// TIA Portal V17 export
// export: Created 2022-07-20T07:02:32.1719581Z, ExportSetting WithDefaults, DisplayName Totally Integrated Automation Portal, DisplayVersion V17, DisplayName TIA Portal Openness, DisplayVersion V17, DisplayName TIA Portal Version Control Interface, DisplayVersion V17, DisplayName SINAMICS Startdrive Advanced, DisplayVersion V17, DisplayName SINAMICS Startdrive G130, G150, S120, S150, SINAMICS MV, S210, DisplayVersion V17, DisplayName SINAMICS Startdrive G110M, G120, G120C, G120D, G120P, G115D, DisplayVersion V17, DisplayName STEP 7 Professional, DisplayVersion V17, DisplayName STEP 7 Safety, DisplayVersion V17, DisplayName WinCC Advanced, DisplayVersion V17
FUNCTION_BLOCK "FB11008_CamTrack"   // FB11008, LAD
{ S7_Optimized_Access := 'TRUE' }
VERSION : 0.1
// stored: AutoNumber false, IsIECCheckEnabled false, IsRetainMemResEnabled false, MemoryReserve 100, SetENOAutomatically false, UDAEnableTagReadback false
   VAR_INPUT
      Enable { ExternalAccessible := 'False'; ExternalVisible := 'False'; ExternalWritable := 'False'} : Bool;
      Cam { ExternalAccessible := 'False'; ExternalVisible := 'False'; ExternalWritable := 'False'} : Array[1..32] of TO_CamTrack_Struct_CamData;
      TimeAdjustmentDown { ExternalAccessible := 'False'; ExternalVisible := 'False'; ExternalWritable := 'False'} : Real;
      TimeAdjustmentUp { ExternalAccessible := 'False'; ExternalVisible := 'False'; ExternalWritable := 'False'} : Real;
   END_VAR
   VAR_OUTPUT
      Error { ExternalAccessible := 'False'; ExternalVisible := 'False'; ExternalWritable := 'False'} : Bool;
      Synchronous : Bool;
      Command { ExternalAccessible := 'False'; ExternalVisible := 'False'; ExternalWritable := 'False'} : Bool;
   END_VAR
   VAR_IN_OUT
      CamTrack : TO_CamTrack;
   END_VAR
   VAR
      instMC_CAMTRACK { ExternalAccessible := 'False'; ExternalVisible := 'False'; ExternalWritable := 'False'} : MC_CAMTRACK;
      R_TRIG_Enable { S7_SetPoint := 'True'} : R_TRIG;
      statNbPoint { S7_SetPoint := 'True'} : UInt;
   END_VAR
BEGIN

REGION Network 1 (SCL): Comments
   //==========================================================================================
   // SIEMENS SAS      RC-FR DI FA APC
   //------------------------------------------------------------------------------------------
   // Restrictions:    TIA V16 and more
   // Requirements:    S7-1500T + MGI library
   // Functionality:   This function block manage a cam track
   //------------------------------------------------------------------------------------------
   // Change log table:
   // Version      Date        Expert in charge    Changes applied
   // 01.00.01     09.06.2020  RTO                 First released version
   //==========================================================================================
END_REGION

REGION Network 2 (SCL): First Scan
   IF "FirstScan" THEN
       ;
   END_IF;
END_REGION

REGION Network 3 (SCL): Edge Signals & Timers
   REGION EDGE SIGNALS
       #R_TRIG_Enable(CLK := #Enable);
   END_REGION

   REGION TIMERS
   END_REGION
END_REGION

REGION Network 4 (SCL): Parameters management
   #CamTrack.Parameter.OnCompensation := #TimeAdjustmentDown;
   #CamTrack.Parameter.OffCompensation := #TimeAdjustmentUp;

   IF #R_TRIG_Enable.Q THEN
       FOR #statNbPoint := 1 TO 32 DO
           #CamTrack.Parameter.Cam[#statNbPoint].Existent := #Cam[#statNbPoint].Existent;
           #CamTrack.Parameter.Cam[#statNbPoint].Duration := #Cam[#statNbPoint].Duration;
           #CamTrack.Parameter.Cam[#statNbPoint].OnPosition := #Cam[#statNbPoint].OnPosition;
           #CamTrack.Parameter.Cam[#statNbPoint].OffPosition := #Cam[#statNbPoint].OffPosition;
       END_FOR;
   END_IF;
END_REGION

REGION Network 5: Manage a cam track
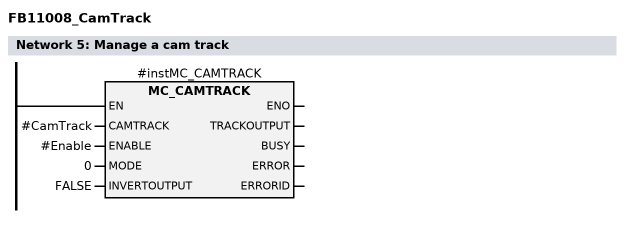
   RUNG wire#powerrail
      #instMC_CAMTRACK.MC_CAMTRACK(CamTrack := #CamTrack, Enable := #Enable, Mode := 0, InvertOutput := FALSE, TrackOutput =>, Busy =>, Error =>, ErrorId =>)
   END_RUNG
   // the same network as SCL:
   #instMC_CAMTRACK(CamTrack := #CamTrack, Enable := #Enable, Mode := 0, InvertOutput := FALSE);   // MC_CAMTRACK
END_REGION

REGION Network 6 (SCL): Manage output
   #Command := #instMC_CAMTRACK.TrackOutput;
   #Synchronous := #CamTrack.StatusWord.%X0;
END_REGION
END_FUNCTION_BLOCK
